# EPICS substitutions: TektronixOscSup/tektronixOsc.substitutions
global{
    CHANNEL_SCAN="\$(CHANNEL_SCAN=5 second)",
    MEASURE_SCAN="\$(MEASURE_SCAN=Passive)"
}

file tektronixOsc_general.template {
    pattern
        {P, PORT}

        {$(P), $(PORT)}
}

file tektronixOsc_channel.template {
    pattern
        {P, PORT, CHANNEL}

        {$(P), $(PORT), 1}
        {$(P), $(PORT), 2}
        {$(P), $(PORT), 3}
        {$(P), $(PORT), 4}
}
